PROGRAM MAIN
VAR
	a:INT;
	b:INT;
	c:INT;
	add1:FB_ADD;
END_VAR

add1(in1:=a , in2:=b , out=>c );

END_PROGRAM

(* stored: Version 1.1.0.1, ProductVersion 3.1.4024.3
   POU MAIN: Id {1c238a28-9b6b-4667-bdaa-7e6877293de4}, SpecialFunc None *)
